% RSLogix 500 project LAB1.RSS, saved by version 8.10.00.30 %
PROJECT "LAB1"    % processor: Bul.1763 MicroLogix 1100 Series A %

PROGRAM FILES
  LAD 2   12 rungs

DATA FILES
  O0 OUTPUT  4 elements
  I1 INPUT  6 elements
  S2 STATUS  66 elements
  B3 BINARY  1 elements
  T4 TIMER  2 elements
  C5 COUNTER  2 elements
  R6 CONTROL  1 elements
  N7 INTEGER  1 elements
  F8 FLOAT  1 elements

LADDER 2
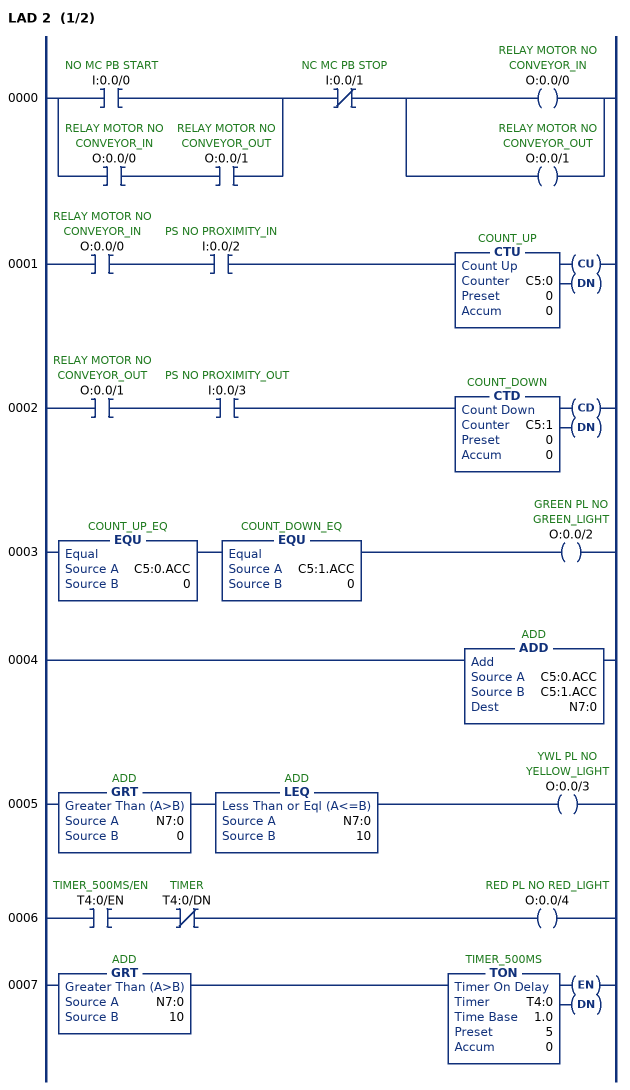
% Rung: 0 %
SOR BST XIC I:0.0/0 NXB XIC O:0.0/0 XIC O:0.0/1 BND XIO I:0.0/1 BST OTE O:0.0/0 NXB OTE O:0.0/1 BND EOR
%   I:0.0/0  START  "NO MC PB" %
%   O:0.0/0  CONVEYOR_IN  "RELAY MOTOR NO" %
%   O:0.0/1  CONVEYOR_OUT  "RELAY MOTOR NO" %
%   I:0.0/1  STOP  "NC MC PB" %
% Rung: 1 %
SOR XIC O:0.0/0 XIC I:0.0/2 CTU C5:0 0 0 EOR
%   O:0.0/0  CONVEYOR_IN  "RELAY MOTOR NO" %
%   I:0.0/2  PROXIMITY_IN  "PS NO" %
%   C5:0  COUNT_UP %
% Rung: 2 %
SOR XIC O:0.0/1 XIC I:0.0/3 CTD C5:1 0 0 EOR
%   O:0.0/1  CONVEYOR_OUT  "RELAY MOTOR NO" %
%   I:0.0/3  PROXIMITY_OUT  "PS NO" %
%   C5:1  COUNT_DOWN %
% Rung: 3 %
SOR EQU C5:0.ACC 0 EQU C5:1.ACC 0 OTE O:0.0/2 EOR
%   C5:0.ACC  COUNT_UP_EQ %
%   C5:1.ACC  COUNT_DOWN_EQ %
%   O:0.0/2  GREEN_LIGHT  "GREEN PL NO" %
% Rung: 4 %
SOR ADD C5:0.ACC C5:1.ACC N7:0 EOR
%   C5:0.ACC  COUNT_UP_EQ %
%   C5:1.ACC  COUNT_DOWN_EQ %
%   N7:0  ADD %
% Rung: 5 %
SOR GRT N7:0 0 LEQ N7:0 10 OTE O:0.0/3 EOR
%   N7:0  ADD %
%   O:0.0/3  YELLOW_LIGHT  "YWL PL NO" %
% Rung: 6 %
SOR XIC T4:0/EN XIO T4:0/DN OTE O:0.0/4 EOR
%   T4:0  TIMER_500MS %
%   T4:0/DN  TIMER %
%   O:0.0/4  RED_LIGHT  "RED PL NO" %
% Rung: 7 %
SOR GRT N7:0 10 TON T4:0 1.0 5 0 EOR
%   N7:0  ADD %
%   T4:0  TIMER_500MS %

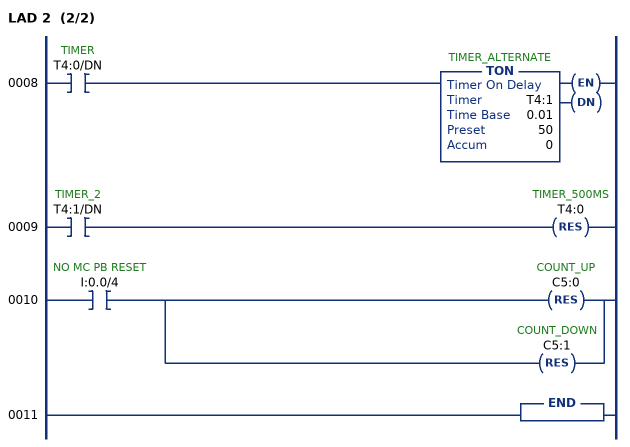
% Rung: 8 %
SOR XIC T4:0/DN TON T4:1 0.01 50 0 EOR
%   T4:0/DN  TIMER %
%   T4:1  TIMER_ALTERNATE %
% Rung: 9 %
SOR XIC T4:1/DN RES T4:0 EOR
%   T4:1/DN  TIMER_2 %
%   T4:0  TIMER_500MS %
% Rung: 10 %
SOR XIC I:0.0/4 BST RES C5:0 NXB RES C5:1 BND EOR
%   I:0.0/4  RESET  "NO MC PB" %
%   C5:0  COUNT_UP %
%   C5:1  COUNT_DOWN %
% Rung: 11 %
SOR END EOR

OTHER DOCUMENTED ADDRESSES
  B3:0/0  CONVEYOR_BIT

DATA TABLE (non-zero values as saved)
DATA T4
% .PRE .ACC %
% T4:0 % 5 0
% T4:1 % 50 0
